FUNCTION Random : REAL
VAR_STAT
	_nSeed	: INT;
END_VAR
VAR
	_drand	: DRAND;
END_VAR

_drand(seed := _nSeed + 1);
Random := LREAL_TO_REAL(_drand.Num);

END_FUNCTION

(* stored: Version 1.1.0.1
   POU Random: Id {ef94bdce-8d7b-4e94-aee6-dfa953145eda}, SpecialFunc None *)
